// SIMATIC S7-200 project (STEP 7-Micro/WIN), CPU 221 REL 01.10

SYMBOL_TABLE USER1
coc              I0.0
bt_an            I0.1
low              I0.2
high             I0.3
bt_den           I0.4
out              Q0.0
bom              Q0.1
den              Q0.2
END_SYMBOL_TABLE

ORGANIZATION_BLOCK MAIN:OB1
TITLE=PROGRAM COMMENTS
BEGIN
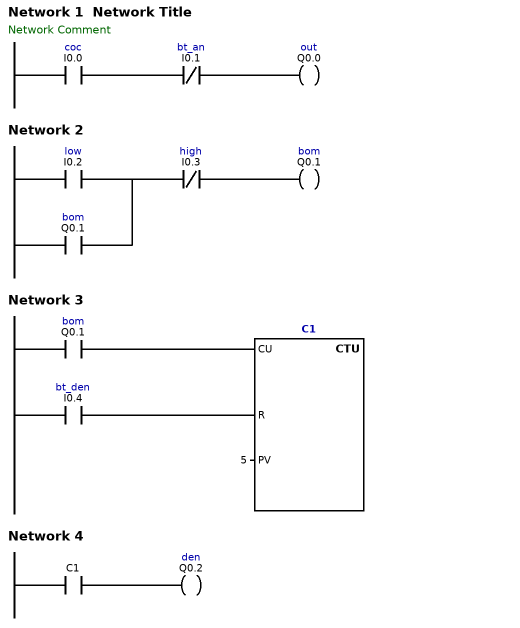
Network 1 // Network Title
// Network Comment
LD     coc:I0.0
AN     bt_an:I0.1
=      out:Q0.0
Network 2
LD     low:I0.2
O      bom:Q0.1
AN     high:I0.3
=      bom:Q0.1
Network 3
LD     bom:Q0.1
LD     bt_den:I0.4
CTU    C1, 5
Network 4
LD     C1
=      den:Q0.2
END_ORGANIZATION_BLOCK
